FUNCTION_BLOCK PolysunBatteryModel (* Client FB for delegating battery model simulations to an external plugin in Polysun. *)
  (* Standard: 61499-2 *)
  (* Version 1.0, 2017-06-18, Marc Jakobi, HTW Berlin *)
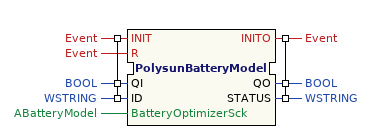
  EVENT_INPUT
    INIT WITH QI, ID; (* Initialization Request *)
    R; (* Release Event *)
  END_EVENT
  EVENT_OUTPUT
    INITO WITH QO, STATUS; (* Initialization Confirm *)
  END_EVENT
  VAR_INPUT
    QI : BOOL; (* Input event qualifier *)
    ID : WSTRING; (* Connection Identifier *)
  END_VAR
  VAR_OUTPUT
    QO : BOOL; (* Output event qualifier *)
    STATUS : WSTRING; (* Service Status *)
  END_VAR
  SOCKETS
    BatteryOptimizerSck : ABatteryModel; (* Link to BatteryOptimizer *)
  END_SOCKETS
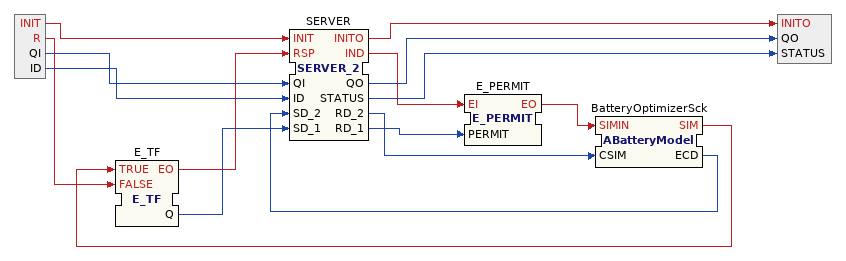
  FBS
    SERVER : SERVER_2;
    E_PERMIT : E_PERMIT;
    E_TF : E_TF;
  END_FBS
  EVENT_CONNECTIONS
    INIT TO SERVER.INIT;
    SERVER.INITO TO INITO;
    SERVER.IND TO E_PERMIT.EI;
    E_PERMIT.EO TO BatteryOptimizerSck.SIMIN;
    BatteryOptimizerSck.SIM TO E_TF.TRUE;
    R TO E_TF.FALSE;
    E_TF.EO TO SERVER.RSP;
  END_CONNECTIONS
  DATA_CONNECTIONS
    QI TO SERVER.QI;
    ID TO SERVER.ID;
    SERVER.QO TO QO;
    SERVER.STATUS TO STATUS;
    SERVER.RD_2 TO BatteryOptimizerSck.CSIM;
    BatteryOptimizerSck.ECD TO SERVER.SD_2;
    SERVER.RD_1 TO E_PERMIT.PERMIT;
    E_TF.Q TO SERVER.SD_1;
  END_CONNECTIONS
END_FUNCTION_BLOCK
